FUNCTION_BLOCK AO_16 (* Composite Function Block Type *)
  (* Standard: 61499-2 *)
  (* Version 0.0, 2018-12-21, 4DIAC-IDE, 4DIAC-Consortium *)
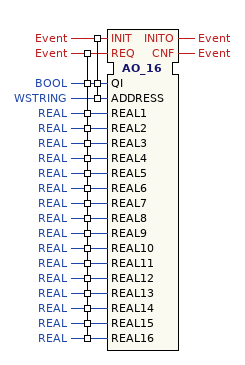
  EVENT_INPUT
    INIT WITH QI, ADDRESS; (* Initialization Request *)
    REQ WITH QI, REAL1, REAL2, REAL3, REAL4, REAL5, REAL6, REAL7, REAL8, REAL9, REAL10, REAL11, REAL12, REAL13, REAL14, REAL15, REAL16; (* Normal Execution Request *)
  END_EVENT
  EVENT_OUTPUT
    INITO; (* Initialization Confirm *)
    CNF; (* Execution Confirmation *)
  END_EVENT
  VAR_INPUT
    QI : BOOL;
    ADDRESS : WSTRING;
    REAL1 : REAL;
    REAL2 : REAL;
    REAL3 : REAL;
    REAL4 : REAL;
    REAL5 : REAL;
    REAL6 : REAL;
    REAL7 : REAL;
    REAL8 : REAL;
    REAL9 : REAL;
    REAL10 : REAL;
    REAL11 : REAL;
    REAL12 : REAL;
    REAL13 : REAL;
    REAL14 : REAL;
    REAL15 : REAL;
    REAL16 : REAL;
  END_VAR
  FBS
    AdressOutputAnalog1 : F_CONCAT;
    AdressOutputAnalog2 : F_CONCAT;
    AdressOutputAnalog3 : F_CONCAT;
    AdressOutputAnalog4 : F_CONCAT;
    AdressOutputAnalog6 : F_CONCAT;
    AdressOutputAnalog7 : F_CONCAT;
    AdressOutputAnalog8 : F_CONCAT;
    AdressOutputAnalog9 : F_CONCAT;
    AdressOutputAnalog10 : F_CONCAT;
    AdressOutputAnalog11 : F_CONCAT;
    AdressOutputAnalog12 : F_CONCAT;
    AdressOutputAnalog13 : F_CONCAT;
    AdressOutputAnalog14 : F_CONCAT;
    AdressOutputAnalog15 : F_CONCAT;
    AdressOutputAnalog16 : F_CONCAT;
    AdressOutputAnalog5 : F_CONCAT;
    PortOutputAnalog1 : WSTRING2WSTRING(IN := :61000);
    PortOutputAnalog2 : WSTRING2WSTRING(IN := :61001);
    PortOutputAnalog4 : WSTRING2WSTRING(IN := :61003);
    PortOutputAnalog3 : WSTRING2WSTRING(IN := :61002);
    PortOutputAnalog5 : WSTRING2WSTRING(IN := :61004);
    PortOutputAnalog6 : WSTRING2WSTRING(IN := :61005);
    PortOutputAnalog7 : WSTRING2WSTRING(IN := :61006);
    PortOutputAnalog8 : WSTRING2WSTRING(IN := :61007);
    PortOutputAnalog9 : WSTRING2WSTRING(IN := :61008);
    PortOutputAnalog10 : WSTRING2WSTRING(IN := :61009);
    PortOutputAnalog11 : WSTRING2WSTRING(IN := :61010);
    PortOutputAnalog12 : WSTRING2WSTRING(IN := :61011);
    PortOutputAnalog13 : WSTRING2WSTRING(IN := :61012);
    PortOutputAnalog14 : WSTRING2WSTRING(IN := :61013);
    PortOutputAnalog15 : WSTRING2WSTRING(IN := :61014);
    PortOutputAnalog16 : WSTRING2WSTRING(IN := :61015);
    CNFOutput16 : E_Merge16;
    InitoOutput16 : E_Merge16;
    OutputAnalog1 : PUBLISH_1;
    OutputAnalog2 : PUBLISH_1;
    OutputAnalog3 : PUBLISH_1;
    OutputAnalog4 : PUBLISH_1;
    OutputAnalog5 : PUBLISH_1;
    OutputAnalog6 : PUBLISH_1;
    OutputAnalog7 : PUBLISH_1;
    OutputAnalog8 : PUBLISH_1;
    OutputAnalog9 : PUBLISH_1;
    OutputAnalog10 : PUBLISH_1;
    OutputAnalog11 : PUBLISH_1;
    OutputAnalog12 : PUBLISH_1;
    OutputAnalog13 : PUBLISH_1;
    OutputAnalog14 : PUBLISH_1;
    OutputAnalog15 : PUBLISH_1;
    OutputAnalog16 : PUBLISH_1;
  END_FBS
  EVENT_CONNECTIONS
    PortOutputAnalog1.CNF TO AdressOutputAnalog1.REQ;
    INIT TO PortOutputAnalog1.REQ;
    PortOutputAnalog2.CNF TO AdressOutputAnalog2.REQ;
    INIT TO PortOutputAnalog2.REQ;
    INIT TO PortOutputAnalog3.REQ;
    PortOutputAnalog3.CNF TO AdressOutputAnalog3.REQ;
    INIT TO PortOutputAnalog4.REQ;
    INIT TO AdressOutputAnalog4.REQ;
    INIT TO PortOutputAnalog5.REQ;
    PortOutputAnalog5.CNF TO AdressOutputAnalog5.REQ;
    INIT TO PortOutputAnalog6.REQ;
    PortOutputAnalog6.CNF TO AdressOutputAnalog6.REQ;
    INIT TO PortOutputAnalog7.REQ;
    PortOutputAnalog7.CNF TO AdressOutputAnalog7.REQ;
    INIT TO PortOutputAnalog8.REQ;
    INIT TO PortOutputAnalog9.REQ;
    PortOutputAnalog9.CNF TO AdressOutputAnalog9.REQ;
    INIT TO PortOutputAnalog10.REQ;
    PortOutputAnalog10.CNF TO AdressOutputAnalog10.REQ;
    INIT TO PortOutputAnalog11.REQ;
    PortOutputAnalog11.CNF TO AdressOutputAnalog11.REQ;
    INIT TO PortOutputAnalog12.REQ;
    PortOutputAnalog12.CNF TO AdressOutputAnalog12.REQ;
    INIT TO PortOutputAnalog13.REQ;
    PortOutputAnalog13.CNF TO AdressOutputAnalog13.REQ;
    INIT TO PortOutputAnalog14.REQ;
    PortOutputAnalog14.CNF TO AdressOutputAnalog14.REQ;
    INIT TO PortOutputAnalog16.REQ;
    INIT TO PortOutputAnalog15.REQ;
    PortOutputAnalog15.CNF TO AdressOutputAnalog15.REQ;
    PortOutputAnalog16.CNF TO AdressOutputAnalog16.REQ;
    PortOutputAnalog8.CNF TO AdressOutputAnalog8.REQ;
    CNFOutput16.EO TO CNF;
    InitoOutput16.EO TO INITO;
    OutputAnalog1.INITO TO InitoOutput16.EI1;
    OutputAnalog3.INITO TO InitoOutput16.EI3;
    OutputAnalog5.INITO TO InitoOutput16.EI5;
    OutputAnalog7.INITO TO InitoOutput16.EI7;
    OutputAnalog8.INITO TO InitoOutput16.EI8;
    OutputAnalog9.INITO TO InitoOutput16.EI9;
    OutputAnalog10.INITO TO InitoOutput16.EI10;
    OutputAnalog11.INITO TO InitoOutput16.EI11;
    OutputAnalog12.INITO TO InitoOutput16.EI12;
    OutputAnalog13.INITO TO InitoOutput16.EI13;
    OutputAnalog14.INITO TO InitoOutput16.EI14;
    OutputAnalog15.INITO TO InitoOutput16.EI15;
    OutputAnalog16.INITO TO InitoOutput16.EI16;
    OutputAnalog1.CNF TO CNFOutput16.EI1;
    OutputAnalog2.CNF TO CNFOutput16.EI2;
    OutputAnalog3.CNF TO CNFOutput16.EI3;
    OutputAnalog5.CNF TO CNFOutput16.EI5;
    OutputAnalog7.CNF TO CNFOutput16.EI7;
    OutputAnalog8.CNF TO CNFOutput16.EI8;
    OutputAnalog9.CNF TO CNFOutput16.EI9;
    OutputAnalog10.CNF TO CNFOutput16.EI10;
    OutputAnalog11.CNF TO CNFOutput16.EI11;
    OutputAnalog12.CNF TO CNFOutput16.EI12;
    OutputAnalog13.CNF TO CNFOutput16.EI13;
    OutputAnalog14.CNF TO CNFOutput16.EI14;
    OutputAnalog15.CNF TO CNFOutput16.EI15;
    OutputAnalog16.CNF TO CNFOutput16.EI16;
    AdressOutputAnalog1.CNF TO OutputAnalog1.REQ;
    AdressOutputAnalog2.CNF TO OutputAnalog2.REQ;
    AdressOutputAnalog4.CNF TO OutputAnalog4.REQ;
    AdressOutputAnalog3.CNF TO OutputAnalog3.REQ;
    AdressOutputAnalog6.CNF TO OutputAnalog6.REQ;
    AdressOutputAnalog5.CNF TO OutputAnalog5.REQ;
    AdressOutputAnalog8.CNF TO OutputAnalog8.REQ;
    AdressOutputAnalog7.CNF TO OutputAnalog7.REQ;
    AdressOutputAnalog9.CNF TO OutputAnalog9.REQ;
    AdressOutputAnalog10.CNF TO OutputAnalog10.REQ;
    AdressOutputAnalog11.CNF TO OutputAnalog11.REQ;
    AdressOutputAnalog12.CNF TO OutputAnalog12.REQ;
    AdressOutputAnalog13.CNF TO OutputAnalog13.REQ;
    AdressOutputAnalog14.CNF TO OutputAnalog14.REQ;
    AdressOutputAnalog16.CNF TO OutputAnalog16.REQ;
    AdressOutputAnalog15.CNF TO OutputAnalog15.REQ;
    INIT TO OutputAnalog1.INIT;
    INIT TO OutputAnalog4.INIT;
    INIT TO OutputAnalog3.INIT;
    INIT TO OutputAnalog5.INIT;
    INIT TO OutputAnalog6.INIT;
    INIT TO OutputAnalog8.INIT;
    INIT TO OutputAnalog7.INIT;
    INIT TO OutputAnalog9.INIT;
    INIT TO OutputAnalog10.INIT;
    INIT TO OutputAnalog11.INIT;
    INIT TO OutputAnalog12.INIT;
    INIT TO OutputAnalog13.INIT;
    INIT TO OutputAnalog14.INIT;
    INIT TO OutputAnalog15.INIT;
    INIT TO OutputAnalog16.INIT;
    REQ TO OutputAnalog1.REQ;
    REQ TO OutputAnalog2.REQ;
    REQ TO OutputAnalog3.REQ;
    REQ TO OutputAnalog4.REQ;
    REQ TO OutputAnalog5.REQ;
    REQ TO OutputAnalog6.REQ;
    REQ TO OutputAnalog8.REQ;
    REQ TO OutputAnalog7.REQ;
    REQ TO OutputAnalog9.REQ;
    REQ TO OutputAnalog10.REQ;
    REQ TO OutputAnalog11.REQ;
    REQ TO OutputAnalog12.REQ;
    REQ TO OutputAnalog14.REQ;
    REQ TO OutputAnalog13.REQ;
    REQ TO OutputAnalog16.REQ;
    REQ TO OutputAnalog15.REQ;
    OutputAnalog2.INITO TO InitoOutput16.EI2;
    INIT TO OutputAnalog2.INIT;
    OutputAnalog4.CNF TO CNFOutput16.EI4;
    OutputAnalog4.INITO TO InitoOutput16.EI4;
    OutputAnalog6.INITO TO InitoOutput16.EI6;
    OutputAnalog6.CNF TO CNFOutput16.EI6;
  END_CONNECTIONS
  DATA_CONNECTIONS
    ADDRESS TO AdressOutputAnalog1.IN1;
    ADDRESS TO AdressOutputAnalog2.IN1;
    ADDRESS TO AdressOutputAnalog3.IN1;
    ADDRESS TO AdressOutputAnalog4.IN1;
    ADDRESS TO AdressOutputAnalog5.IN1;
    ADDRESS TO AdressOutputAnalog6.IN1;
    ADDRESS TO AdressOutputAnalog7.IN1;
    ADDRESS TO AdressOutputAnalog8.IN1;
    ADDRESS TO AdressOutputAnalog9.IN1;
    ADDRESS TO AdressOutputAnalog10.IN1;
    ADDRESS TO AdressOutputAnalog11.IN1;
    ADDRESS TO AdressOutputAnalog12.IN1;
    ADDRESS TO AdressOutputAnalog15.IN1;
    ADDRESS TO AdressOutputAnalog16.IN1;
    PortOutputAnalog1.OUT TO AdressOutputAnalog1.IN2;
    PortOutputAnalog2.OUT TO AdressOutputAnalog2.IN2;
    PortOutputAnalog3.OUT TO AdressOutputAnalog3.IN2;
    PortOutputAnalog4.OUT TO AdressOutputAnalog4.IN2;
    PortOutputAnalog5.OUT TO AdressOutputAnalog5.IN2;
    PortOutputAnalog6.OUT TO AdressOutputAnalog6.IN2;
    PortOutputAnalog8.OUT TO AdressOutputAnalog8.IN2;
    PortOutputAnalog7.OUT TO AdressOutputAnalog7.IN2;
    PortOutputAnalog10.OUT TO AdressOutputAnalog10.IN2;
    PortOutputAnalog9.OUT TO AdressOutputAnalog9.IN2;
    PortOutputAnalog11.OUT TO AdressOutputAnalog11.IN2;
    PortOutputAnalog12.OUT TO AdressOutputAnalog12.IN2;
    PortOutputAnalog13.OUT TO AdressOutputAnalog13.IN2;
    PortOutputAnalog14.OUT TO AdressOutputAnalog14.IN2;
    PortOutputAnalog15.OUT TO AdressOutputAnalog15.IN2;
    PortOutputAnalog16.OUT TO AdressOutputAnalog16.IN2;
    ADDRESS TO AdressOutputAnalog13.IN1;
    ADDRESS TO AdressOutputAnalog14.IN1;
    AdressOutputAnalog1.OUT TO OutputAnalog1.ID;
    AdressOutputAnalog2.OUT TO OutputAnalog2.ID;
    AdressOutputAnalog4.OUT TO OutputAnalog4.ID;
    AdressOutputAnalog3.OUT TO OutputAnalog3.ID;
    AdressOutputAnalog7.OUT TO OutputAnalog7.ID;
    AdressOutputAnalog5.OUT TO OutputAnalog5.ID;
    AdressOutputAnalog6.OUT TO OutputAnalog6.ID;
    AdressOutputAnalog8.OUT TO OutputAnalog8.ID;
    AdressOutputAnalog10.OUT TO OutputAnalog10.ID;
    AdressOutputAnalog9.OUT TO OutputAnalog9.ID;
    AdressOutputAnalog12.OUT TO OutputAnalog12.ID;
    AdressOutputAnalog11.OUT TO OutputAnalog11.ID;
    AdressOutputAnalog14.OUT TO OutputAnalog14.ID;
    AdressOutputAnalog13.OUT TO OutputAnalog13.ID;
    AdressOutputAnalog16.OUT TO OutputAnalog16.ID;
    AdressOutputAnalog15.OUT TO OutputAnalog15.ID;
    QI TO OutputAnalog1.QI;
    QI TO OutputAnalog2.QI;
    QI TO OutputAnalog3.QI;
    QI TO OutputAnalog4.QI;
    QI TO OutputAnalog5.QI;
    QI TO OutputAnalog6.QI;
    QI TO OutputAnalog7.QI;
    QI TO OutputAnalog8.QI;
    QI TO OutputAnalog9.QI;
    QI TO OutputAnalog10.QI;
    QI TO OutputAnalog11.QI;
    QI TO OutputAnalog12.QI;
    QI TO OutputAnalog13.QI;
    QI TO OutputAnalog14.QI;
    QI TO OutputAnalog15.QI;
    QI TO OutputAnalog16.QI;
    REAL1 TO OutputAnalog1.SD_1;
    REAL2 TO OutputAnalog2.SD_1;
    REAL3 TO OutputAnalog3.SD_1;
    REAL4 TO OutputAnalog4.SD_1;
    REAL5 TO OutputAnalog5.SD_1;
    REAL6 TO OutputAnalog6.SD_1;
    REAL7 TO OutputAnalog7.SD_1;
    REAL8 TO OutputAnalog8.SD_1;
    REAL9 TO OutputAnalog9.SD_1;
    REAL10 TO OutputAnalog10.SD_1;
    REAL11 TO OutputAnalog11.SD_1;
    REAL12 TO OutputAnalog12.SD_1;
    REAL13 TO OutputAnalog13.SD_1;
    REAL14 TO OutputAnalog14.SD_1;
    REAL15 TO OutputAnalog15.SD_1;
    REAL16 TO OutputAnalog16.SD_1;
  END_CONNECTIONS
END_FUNCTION_BLOCK
